{attribute 'qualified_only'}
{attribute 'strict'}
{attribute 'to_string'}
TYPE E_DirectionSelect :
(
    UNDEFINED := -1,
	FORWARD := 0,
    LEFT,
    RIGHT
);
END_TYPE

(* stored: Version 1.1.0.1
   DUT E_DirectionSelect: Id {3dd11271-3c8d-4e73-8679-866791950f66} *)
